(* PLC project Tc2_Utilities.UInt64Add64Ex Demo, tc3-libraries-kb TwinCAT 3.1 *)
(* stored: creationDateTime 2026-05-10T18:00:00, modificationDateTime 2026-05-10T18:00:00 *)

PROGRAM P_Demo_UInt64Add64Ex
  VAR
    rResult : T_ULARGE_INTEGER;  (* UInt64Add64Ex 返回值 *)
    bRun : BOOL;  (* 触发一次调用 *)
    a : T_ULARGE_INTEGER;  (* 测试用本地变量 *)
    b : T_ULARGE_INTEGER;  (* 测试用本地变量 *)
    bOV : BOOL;  (* 测试用本地变量 *)
  END_VAR

            // ============================================================
// Tc2_Utilities.UInt64Add64Ex 演示程序（FUNCTION）
// ============================================================
// 验证步骤：
//   1. 引用 Tc2_Utilities
//   2. 编译 + 登录
//   3. 强制 bRun := TRUE 一个周期
//   4. 在线监视 rResult
// ============================================================

a := ULARGE_INTEGER(16#FFFFFFFF, 16#FFFFFFFF); b := ULARGE_INTEGER(0, 1);
IF bRun THEN
    rResult := UInt64Add64Ex(augend := a, addend := b, bOV := bOV);
    bRun := FALSE;
END_IF;

          
END_PROGRAM
